(* IEC 61131-3 sources: ae-axftcmlib/src, 2 files *)

(* ---- configuration.st ---- *)
USING Simatic;
USING Simatic.Ax.axftcmlib;
//Additionally needed
USING Simatic.Ax.IO.Output;
USING Simatic.Ax.IO.Input;

CONFIGURATION axftcmlibconfig
    TASK Main(Interval := T#100ms, Priority := 1);
    PROGRAM P1 WITH Main: ExampleForAxftcm_Program;

    VAR_GLOBAL
        //All PLC-Variables used
        SortinglineStartingLightbarrier     AT %I200.1 : BOOL;
        SortinglineEndLightbarrier          AT %I200.2 : BOOL;
        SortinglineMotorForConveyor         AT %Q200.0 : BOOL;
        SortinglineCompressor               AT %Q200.1 : BOOL;
        SortinglineValveEjector             AT %Q200.3 : BOOL;
    END_VAR

    VAR_GLOBAL
        //Binoutputs are used to cyclicly write on the PLC-Variables
        //They help with communicating and are used in the axftcmlib
        //ALso available on GitHub as a separate repository (IO)
        CompressorOutputWriter      : BinOutput;
        CylinderOutputWriter        : BinOutput;
        MotorForwardOutputWriter    : BinOutput;
        MotorBackwardsOutputWriter  : BinOutput;

        //BinSignals are used to track inputs from the model
        //ALso included in the IO libraray
        //The Output is inverted because the lightbarrieres return False if they detect something
        StartingLightbarriereReader : BinSignal := (Invert := TRUE);
        EndingLightbarrierReader    : BinSignal := (Invert := TRUE);
        AxisReferenceswitch         : BinSignal;

        //Actual instances of the Elements used in the sortingline
        CompressorClassInstance         :   PneumaticCompressor :=  (ActiveCompressor := CompressorOutputWriter);
        CylinderClassInstance           :   ActuatorTimeBased   :=  (ControlPush      := CylinderOutputWriter);

        //Axis:
        //An Encoder as well as a Timeprovider are needed to gereate the current position of the conveyorbelt
        TimeproviderForAxis             : Timeprovider;
        MotorForAxis                    : MotorFT           := (Forward := MotorForwardOutputWriter, Reverse := MotorBackwardsOutputWriter);
        TimebasedEncoderForAxis         : TimeBasedEncoder  := (Timeprovider := TimeproviderForAxis, EncoderAxis := ConveyorbeltForSortingline, Velocity := 1.0);
        ConveyorbeltForSortingline      : Axis              := (Motor :=  MotorForAxis, Encoder := TimebasedEncoderForAxis, ReferenceSwitch := AxisReferenceswitch);

        //Controlvariables
        Statecounter                    : INT               := (0);

    END_VAR
END_CONFIGURATION

(* ---- program.st ---- *)
USING Simatic;
USING Simatic.Ax.axftcmlib;
//Additionally needed
USING Simatic.Ax.IO.Output;
USING Simatic.Ax.IO.Input;

PROGRAM ExampleForAxftcm_Program
    ///Functrion:
    /// If an element is added to the front lightbarrier, it activates the conveyor
    /// the conveyor moves the piece to the cylinder, where it is pushed into the chute
    VAR_EXTERNAL
        //All global variables used in this Programm have to be "included" as VAR_EXTERNAL
        SortinglineStartingLightbarrier     : BOOL;
        SortinglineEndLightbarrier          : BOOL;
        SortinglineMotorForConveyor         : BOOL;
        SortinglineCompressor               : BOOL;
        SortinglineValveEjector             : BOOL;

        CompressorOutputWriter              : BinOutput;
        CylinderOutputWriter                : BinOutput;
        MotorForwardOutputWriter            : BinOutput;
        MotorBackwardsOutputWriter          : BinOutput;

        StartingLightbarriereReader         : BinSignal;
        EndingLightbarrierReader            : BinSignal;
        AxisReferenceswitch                 : BinSignal;

        CompressorClassInstance             : PneumaticCompressor;
        CylinderClassInstance               : ActuatorTimeBased;

        TimeproviderForAxis                 : Timeprovider;
        MotorForAxis                        : MotorFT;
        TimebasedEncoderForAxis             : TimeBasedEncoder;
        ConveyorbeltForSortingline          : Axis;

        Statecounter                        : INT;
    END_VAR

    VAR
        //Local variables could be added here but note that they cant be monitored
    END_VAR

    ///Reading the state of the lightbarrier every Cycle
    StartingLightbarriereReader.ReadCyclic(SortinglineStartingLightbarrier);
    EndingLightbarrierReader.ReadCyclic(SortinglineEndLightbarrier);

    ///Needs to be called in every cycle
    CylinderClassInstance.RunCyclic();
    ConveyorbeltForSortingline.RunCyclic();

    ///Get and Process the cycletime every cycle
    TimebasedEncoderForAxis.Evaluate();
    TimeproviderForAxis.Evaluate();

    IF Statecounter = 0 AND StartingLightbarriereReader.QRis() THEN
       ConveyorbeltForSortingline.Homing(Position := 0);
        ConveyorbeltForSortingline.MoveAbsolute(Velocity := 1.0, Position := 4150);
        Statecounter := 1;
    END_IF;

    IF Statecounter = 1 AND EndingLightbarrierReader.QRis() THEN
        CompressorClassInstance.PneumaticCompressorOn();
        Statecounter := 2;
    END_IF;

    IF Statecounter = 2 AND EndingLightbarrierReader.QFal() THEN
        CylinderClassInstance.Enable();
        Statecounter := 0;
    END_IF;

    //Actually writing the results onto the PLCs variables
    CylinderOutputWriter.WriteCyclic(Q => SortinglineValveEjector);
    CompressorOutputWriter.WriteCyclic(Q => SortinglineCompressor);
    MotorForwardOutputWriter.WriteCyclic(Q => SortinglineMotorForConveyor);

    ;
END_PROGRAM
